FUNCTION_BLOCK FB_HMI_SERVICES_TIME EXTENDS FB_HMI_COMPONENT
VAR_INPUT
END_VAR
VAR_OUTPUT
END_VAR
VAR_IN_OUT
    fbInstance : FB_TIME;
END_VAR
VAR
    // because GUI_TEMPLATE_TIME is a large height,
    // and because scrolling doesn't seem to work (bug in TC HMI?),
    // we display the GUI_TEMPLATE_TIME twice, with an offset in between 
    nAbsoluteMovementY : INT := -495;
    
    sUtc : STRING;
END_VAR


// update the health & busy states
fbHealthStatus(
    bIsGood     := fbInstance.stat.signal.qos = E_TIME_SIGNAL_QOS.VALID,
    bIsEnabled  := fbInstance.stat.signal.status = E_TIME_SIGNAL_STATUS.CONNECTED);
fbBusyStatus(bIsBusy := FALSE); // never busy

sUtc := LEFT(fbInstance.stat.sUtcTime, 19); 

M_UpdateStatusColor();

END_FUNCTION_BLOCK

(* stored: Version 1.1.0.1, ProductVersion 3.1.4024.14
   POU FB_HMI_SERVICES_TIME: Id {e23eebbf-6ab2-46e1-8d9a-93fd51686b76}, SpecialFunc None *)
